FUNCTION_BLOCK UT_AuxiliaryInputMapping_Type_03_Analog_Ret50perc (* Type 3 Analog_Ret50perc Two way analog - return to centre position *)
  (* Standard: ISO 11783-6; Classification: AUX – ISO 11783-6; Function: All Inputs; Type: UT according to ISO 11783-6; Description: - Type 3 Analog_Ret50perc Two way analog - return to centre position Applicable AUX-N only * maps to IW IW - Input WORD (16 Bit) *)
  (* Version 1.0, 2018-12-05, Jose Cabral *)
  (* Version 1.1, 2022-08-04, Franz Höpfinger, HR Agrartechnik GmbH *)
  (* Version 1.2, 2023-01-05, Franz Höpfinger, HR Agrartechnik GmbH *)
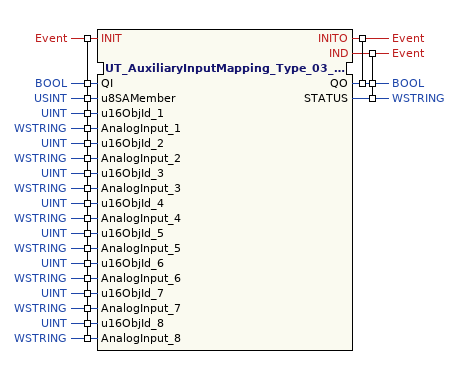
  EVENT_INPUT
    INIT WITH QI, u8SAMember, u16ObjId_1, AnalogInput_1, u16ObjId_2, AnalogInput_2, u16ObjId_3, AnalogInput_3, u16ObjId_4, AnalogInput_4, u16ObjId_5, AnalogInput_5, u16ObjId_6, AnalogInput_6, u16ObjId_7, AnalogInput_7, u16ObjId_8, AnalogInput_8; (* Service Initialization *)
  END_EVENT
  EVENT_OUTPUT
    INITO WITH QO; (* Initialization Confirm *)
    IND WITH QO, STATUS; (* Indication from Resource *)
  END_EVENT
  VAR_INPUT
    QI : BOOL; (* Event Input Qualifier *)
    u8SAMember : USINT := 255; (* Dummy !, set to 255 if in doubt. 0 deactivates FB. *)
    u16ObjId_1 : UINT := 31000; (* Object ID of Input 1 *)
    AnalogInput_1 : WSTRING := "AuxInput_31000"; (* Identifier for Input 1 *)
    u16ObjId_2 : UINT := 31001; (* Object ID of Input 2 *)
    AnalogInput_2 : WSTRING := "AuxInput_31001"; (* Identifier for Input 2 *)
    u16ObjId_3 : UINT := 31002; (* Object ID of Input 3 *)
    AnalogInput_3 : WSTRING := "AuxInput_31002"; (* Identifier for Input 3 *)
    u16ObjId_4 : UINT := 31003; (* Object ID of Input 4 *)
    AnalogInput_4 : WSTRING := "AuxInput_31003"; (* Identifier for Input 4 *)
    u16ObjId_5 : UINT := 31004; (* Object ID of Input 5 *)
    AnalogInput_5 : WSTRING := "AuxInput_31004"; (* Identifier for Input 5 *)
    u16ObjId_6 : UINT := 31005; (* Object ID of Input 6 *)
    AnalogInput_6 : WSTRING := "AuxInput_31005"; (* Identifier for Input 6 *)
    u16ObjId_7 : UINT := 31006; (* Object ID of Input 7 *)
    AnalogInput_7 : WSTRING := "AuxInput_31006"; (* Identifier for Input 7 *)
    u16ObjId_8 : UINT := 31007; (* Object ID of Input 8 *)
    AnalogInput_8 : WSTRING := "AuxInput_31007"; (* Identifier for Input 8 *)
  END_VAR
  VAR_OUTPUT
    QO : BOOL; (* Event Output Qualifier *)
    STATUS : WSTRING; (* Service Status *)
  END_VAR
END_FUNCTION_BLOCK
